# EPICS substitutions: NWPRTXPS/NWPRTXPS-IOC-01App/Db/motor.substitutions
file $(MOTOR)/motorApp/Db/basic_asyn_motor.db {
    pattern {P,    M,         ADDR, DTYP,      PORT, DESC,   EGU,  VELO,  VBAS, ACCL, BDST, BVEL, BACC,    MRES,    ERES,  PREC, DHLM, DLLM, INIT, DIR}
         {"\$(P)", "\$(M)", 0, "asynMotor", "\$(XPS_PORT)", "DESC",    "mm",   "100",   "0",  "1",    0,    1,   0,   "\$(MRES)",   "\$(ERES)",    3,   "360",   "0",  "", "Pos"}
}

file "$(MOTOR)/db/XPS_extra.db"{
    pattern {P,     R,  PORT,  ADDR}
        {"\$(P)",  m1, "\$(XPS_PORT)",  0}
}
